FUNCTION F_PVOID_RTN : PVOID
VAR_INPUT
	stArg : ST_Arg;
END_VAR
VAR_STAT
	sysVar_Info : __SYSTEM.VAR_INFO;
END_VAR

sysVar_Info := __VARINFO(F_PVOID_RTN);
IF stArg.TypeClass = sysVar_Info.TypeClass THEN 
	F_PVOID_RTN := stArg.pValue;
	END_IF

END_FUNCTION

(* stored: Version 1.1.0.1, ProductVersion 3.1.4024.4
   POU F_PVOID_RTN: Id {b81b3b5f-5a7f-44b3-81ae-f7a4c81ab71f}, SpecialFunc None *)
